{attribute 'hide_all_locals'}
FUNCTION_BLOCK EcMasterState IMPLEMENTS IEcTask
VAR_INPUT
END_VAR
VAR_OUTPUT
END_VAR
VAR
	iState : INT;
	getMasterState : Tc2_EtherCAT.FB_EcGetMasterState;
	_execute: BOOL;
	_done: BOOL;
	_busy: BOOL;
	_error: BOOL;
	
END_VAR

CASE iState OF
	0:
		IF _execute THEN
			_done := FALSE;
			_busy := TRUE;
			_error := FALSE;
			getMasterState.bExecute := TRUE;
			IF getMasterState.bBusy THEN
				iState := 10;
				_execute := false;
			END_IF
		END_IF
	10:
		IF NOT getMasterState.bBusy THEN
			IF NOT getMasterState.bError THEN
				_done := TRUE;
			ELSE
				_error := TRUE;
			END_IF
			_busy := FALSE;
			getMasterState.bExecute := FALSE;
			iState := 0;
		END_IF
END_CASE

getMasterState(sNetId := Tc2_System.F_CreateAmsNetId(nIds := NetId));

{warning 'add method implementation '}
METHOD Abort : BOOL
getMasterState.bExecute := FALSE;
_busy := FALSE;
_execute := FALSE;
Abort := TRUE;
iState := 0;
END_METHOD

{warning 'add property implementation'}
PROPERTY Busy : BOOL
GET
Busy := _busy;
END_GET
END_PROPERTY

{warning 'add property implementation'}
PROPERTY Done : BOOL
GET
Done := _done;
END_GET
END_PROPERTY

{warning 'add property implementation'}
PROPERTY Error : BOOL
GET
Error := _error;
END_GET
END_PROPERTY

{warning 'add method implementation '}
METHOD Execute : BOOL
IF NOT getMasterState.bBusy THEN
	Execute := _execute := TRUE;
END_IF
END_METHOD

PROPERTY MasterState : word
GET
MasterState := getMasterState.state;
END_GET
END_PROPERTY

{warning 'add property implementation'}
PROPERTY NetID : amsnetid
GET
NetID := _netId;
END_GET
SET
_netId := NetID;
END_SET
END_PROPERTY

END_FUNCTION_BLOCK

(* stored: Version 1.1.0.1, ProductVersion 3.1.4024.11
   POU EcMasterState: Id {3609d461-0de1-4e7e-8e58-79ac738134c4}, SpecialFunc None
   Method Abort: Id {a94af2ee-47ba-4f21-a620-1155aaf081be}
   Property Busy: Id {c86c0f33-2698-4f06-8bfe-638a7a9e36f3}
   Get Get: Id {0ac9899b-742a-4112-8d89-03d9ab3a849d}
   Property Done: Id {bb76d6f4-3f3b-41a4-8c69-c5dd6b0c2748}
   Get Get: Id {7a8de72d-9e55-4e8e-b063-94038cb0e0ad}
   Property Error: Id {e899f1f4-382b-40f8-9bad-62bd6fb7cbd5}
   Get Get: Id {ac004b05-e046-4c57-9ee6-a741f4b60038}
   Method Execute: Id {0b99a093-a365-4c6e-8af4-3a4f98f1cecb}
   Property MasterState: Id {722d365c-a1e9-4bcf-97dc-972aa8953e80}
   Get Get: Id {245ba7d2-689d-40a7-a076-06b6e28ecba9}
   Property NetID: Id {ade085ad-1c54-4ca5-85ac-5595386b4a10}
   Get Get: Id {7b0d4fa8-9f39-442b-b308-1809b77cd043}
   Set Set: Id {6d50682b-2831-48f6-aab1-501fdd97ca57} *)
